(* CODESYS project ExtractAnyString.library
   Author: Piotr Pawlowski
   Version: 1.0.0.0
   Company: Marden Edwards
   Title: Extrac String
   Placeholder: EXTRACT
   LanguageModelAttribute: qualified-access-only
   DefaultNamespace: EXTRACT
   DocFormat: TcDocGen

Project tree, tasks and I/O mapping:
  libraries: Tc2_Standard, * (Beckhoff Automation GmbH); Tc2_System, * (Beckhoff Automation GmbH); Tc2_Utilities, * (Beckhoff Automation GmbH)
  DUTs/
    String/
      data type E_ExtrMode
      data type T_Char
      data type T_LongSTRING
  GVLs/
  POUs/
    String FB/
      function block FB_ExtractAnyString [ST]
      function block FB_ExtractString [ST]
    Strings FUN/
      function F_ReplaceLongSingleChar [ST]
  Version/
    global variables Global_Version
*)

// DUTs/String/E_ExtrMode
{attribute 'qualified_only'}
{attribute 'strict'}
TYPE E_ExtrMode :
(
	WITHIDENT,						//extract with ident and dont purge left side string
	WITHIDENT_PURGE,				//extract with ident and purge left side string
	WITHOUTIDENT,					//extract with ident and dont purge left side string, both ident left in origin string 
	WITHOUTIDENT_PURGE,				//extract with ident and purge left side string, only sufix ident left in origin string
	WITHOUTIDENT_REMIDENT,			//extract with ident and dont purge left side string, no ident left in origin string
	WITHOUTIDENT_REMIDENT_PURGE		//extract with ident and purge left side string, no ident left in origin string
);
END_TYPE

// DUTs/String/T_Char
TYPE T_Char : STRING[1];
END_TYPE

// DUTs/String/T_LongSTRING
TYPE T_LongSTRING : STRING(1023);
END_TYPE

// Version/Global_Version
{attribute 'TcGenerated'}
{attribute 'no-analysis'}
{attribute 'linkalways'}
// This function has been automatically generated from the project information.
VAR_GLOBAL CONSTANT
	{attribute 'const_non_replaced'}
	stLibVersion_Extrac_String : ST_LibVersion := (iMajor := 1, iMinor := 0, iBuild := 0, iRevision := 0, nFlags := 0, sVersion := '1.0.0.0');
END_VAR

// POUs/String FB/FB_ExtractAnyString
// Extracts a sub-string defined by prefix and suffix 
// Works in one cycle but as FB to not use stack memore due to LongString data defined
FUNCTION_BLOCK FB_ExtractAnyString
VAR_INPUT
	bExtractData			: BOOL;			(* set TRUE to remove prefix and suffix from strData *)
	nExtractChars			: UDINT;			(* if suffix is blank, number of data chars to extract *)
	sPrefix					: T_LongSTRING;	(* prefix string extended from T_MaxString to T_LongSTRING *)
	sSuffix					: T_LongSTRING;	(* suffix string extended from T_MaxString to T_LongSTRING *)
	bIgnoreCase				: BOOL;
	eExtractMode			: E_ExtrMode	:= E_ExtrMode.WITHOUTIDENT_REMIDENT;
	//bIncludeIdentifiers	: BOOL;
END_VAR
VAR_IN_OUT
	sDataString				: T_LongSTRING;	(* string to be searched *)
END_VAR
VAR_OUTPUT
	bStringFound			: BOOL;			(* TRUE = sub-string with matching prefix/suffix found *)
	sExtractedString		: T_LongSTRING;	(* extracted data *)
	nExtractedStringPos		: UDINT;			(* start pos of extracted string in strString *)
	nExtractedStringLen		: UDINT;
	nDataStringLen			: UDINT;
END_VAR
VAR
	
	//_rtExecute			: R_trig;
	
	_nExtractChars			: UDINT;
	_sPrefix				: T_LongSTRING;	(* prefix string *)
	_sSuffix				: T_LongSTRING;	(* suffix string *)
	_sDataString			: T_LongSTRING;	(* string to be searched *)
	
	_bIncludeIdentifiers	: BOOL;
	_bPurgeFullString		: BOOL;
	
	_nDataStringLen			: UDINT;
	_nPrefixLen				: UDINT;
	_nSuffixLen				: UDINT;
	
	_bPrefixFound			: BOOL;
	_bSuffixFound			: BOOL;
	
	_bPrefixIndex			: UDINT;
	_bTempSuffixIndex		: UDINT;
	_bSuffixIndex			: UDINT;
	
	_nStartDataPos			: UDINT;
	_nAbsolutDataPos		: UDINT;
	_nEndDataPos			: UDINT;
	_nExtractedDataLen		: UDINT;
	
	_nTerminatePos			: UDINT;
END_VAR

//	EXTRWITHIDENT						//extract with ident and dont purge left side string
//	EXTRWITHIDENT_PURGE					//extract with ident and purge left side string
//	EXTRWITHOUTIDENT					//extract with ident and dont purge left side string, both ident left in origin string 
//	EXTRWITHOUTIDENT_PURGE				//extract with ident and purge left side string, only sufix ident left in origin string
//	EXTRWITHOUTIDENT_REMIDENT			//extract with ident and dont purge left side string, no ident left in origin string
//	EXTRWITHOUTIDENT_REMIDENT_PURGE		//extract with ident and purge left side string, no ident left in origin string

//====================================================================================	
IF 	eExtractMode = E_ExtrMode.WITHIDENT 			OR 
	eExtractMode = E_ExtrMode.WITHIDENT_PURGE 	THEN
	
	_bIncludeIdentifiers	:= TRUE;
ELSE 
	_bIncludeIdentifiers	:= FALSE;
END_IF

IF 	eExtractMode = E_ExtrMode.WITHIDENT_PURGE 		OR 
	eExtractMode = E_ExtrMode.WITHOUTIDENT_PURGE 	OR 
	eExtractMode = E_ExtrMode.WITHOUTIDENT_REMIDENT_PURGE THEN
	
	_bPurgeFullString	:= LEN2(ADR(sDataString)) = SIZEOF(sDataString)-1;
ELSE 
	_bPurgeFullString	:= FALSE;
END_IF

//====================================================================================	

(* rising edge of bExecute *)
//_rtExecute(CLK := bExtractData);

//IF _rtExecute.Q THEN
	
//====================================================================================	
	bStringFound 		:= FALSE;
	
	_sDataString 		:= '';
	_sPrefix 			:= '';
	_sSuffix 			:= '';
	
	_bPrefixFound		:= FALSE;
	_bSuffixFound		:= FALSE;
		
	_bPrefixIndex		:= 0;
	_bSuffixIndex		:= 0;
		
	_nStartDataPos		:= 0;
	_nAbsolutDataPos	:= 0;
	_nEndDataPos		:= 0;
	//_ExtractedDataLen	:= 0;
	
	 (*calc string lengths *)
	_nDataStringLen 	:= LEN2(ADR(sDataString));
	_nPrefixLen 		:= LEN2(ADR(sPrefix));
	_nSuffixLen 		:= LEN2(ADR(sSuffix));
	
	_nExtractChars:= LIMIT(0, nExtractChars, _nDataStringLen);
	
	(*clear outputs*)
	nExtractedStringPos	:= 0;
	nExtractedStringLen	:= 0;
	nDataStringLen		:= _nDataStringLen;

//====================================================================================	
	
	(* matching for Prefix and Suffix is case-sesnsitive - worsk only with T_MaxString *)
	IF bIgnoreCase AND 
		_nDataStringLen < 256 	AND 
		_nPrefixLen < 256 		AND 
		_nSuffixLen < 256 		THEN
		
		(* internal comparators are all converted to lower case *)
		_sDataString 	:= F_ToLCase(sDataString);
		_sPrefix 		:= F_ToLCase(sPrefix);
		_sSuffix 		:= F_ToLCase(sSuffix);
		
	ELSE
		(* internal comparators are not changed *)
		_sDataString 	:= sDataString;
		_sPrefix 		:= sPrefix;
		_sSuffix 		:= sSuffix;
	END_IF

//====================================================================================	

	IF _nPrefixLen = 0 AND  _nExtractChars > 0 THEN
		
		_bPrefixIndex		:= 1;
		_nStartDataPos		:= 1;
		nExtractedStringPos := 1;
		
	ELSIF _nPrefixLen > 0 THEN		//if _nPrefixLen = 0 then _bPrefixIndex and _StartDataPos remains 0 from init state
		
		_bPrefixIndex	:= FIND2(ADR(_sDataString), ADR(_sPrefix));		//find search only if prefix declared on the input
	
		IF _bPrefixIndex > 0 THEN		//_bPrefixIndex as result form find can be onlu positive range
			
			_bPrefixFound := TRUE;		// _bPrefixFound guarantee _StartDataPos > 0
			_nStartDataPos 	:= SEL(_bIncludeIdentifiers, _bPrefixIndex + _nPrefixLen, _bPrefixIndex);
			_nAbsolutDataPos	:= _bPrefixIndex + _nPrefixLen;
			
			nExtractedStringPos := _nStartDataPos;
		END_IF
	END_IF	
	
//====================================================================================		

	IF _nSuffixLen = 0 AND  _nExtractChars > 0 THEN //IF only nExtractChars is declared THEN _EndDataPos pointing on elemnt determinated by nExtractChars or on last elemnt OF DataString
		
		_bSuffixIndex := _bPrefixIndex + _nPrefixLen + _nExtractChars;
		_nEndDataPos := MIN(_bSuffixIndex, _nDataStringLen);
		
		IF _nEndDataPos > _nStartDataPos THEN  // check if both pointers not point on last DataString elemnt
			_bSuffixFound := TRUE;	// _bSuffixFound guarantee _EndDataPos > 0 and found after _StartDataPos
		END_IF
		
	ELSIF _nSuffixLen > 0 THEN // if _nSuffixLen declared, then ignor nExtractChars and search for find sufix position using 
		
		// Include Sufix change shift if onle Prfix was found >> SEL(_bPrefixFound, 0, _StartDataPos - 1)
		_bTempSuffixIndex	:= FIND2(ADR(_sDataString) + SEL(_bPrefixFound, 0, _nAbsolutDataPos - 1), ADR(_sSuffix)); //find search only if sufix declared on the input and on index after prefix
		IF _bTempSuffixIndex > 0 THEN
			_bSuffixIndex	:= _bTempSuffixIndex + SEL(_bPrefixFound, 0, _nAbsolutDataPos - 1);	//Recalculate Sufix real position if sufix found or _bSuffixIndex remain 0 form init
		END_IF
		
		(*_bTempSuffixIndex gurantee that sufix was search after prefix position so _EndDataPos always greater than _StartDataPos *) 
		IF _bSuffixIndex > 0 THEN
			_bSuffixFound := TRUE;	// _bSuffixFound guarantee _EndDataPos > 0
			_nEndDataPos := SEL(_bIncludeIdentifiers,_bSuffixIndex, _bSuffixIndex + _nSuffixLen);
		END_IF
	END_IF
	
//====================================================================================		
	
	MEMSET(ADR(sExtractedString), 16#00, SIZEOF(sExtractedString));	//Clean sExtractedString area for new data

	IF _bPrefixFound AND _bSuffixFound THEN

		DELETE2(ADR(sDataString), ADR(sExtractedString), SIZEOF(sExtractedString), 
											SIZEOF(sExtractedString) - _nEndDataPos , _nEndDataPos);
		DELETE2(ADR(sExtractedString), ADR(sExtractedString), SIZEOF(sExtractedString), _nStartDataPos -1, 1);
		
	ELSIF _nPrefixLen = 0 AND _nSuffixLen = 0 AND _nExtractChars >= _nEndDataPos THEN		
		
		sExtractedString := sDataString;
		
	ELSIF _nPrefixLen = 0 AND _bSuffixFound THEN		// TO BE CONSIDERED IF WE WANT THIS CONDITION - IT WORKS LIKE LEFT
		
		_nStartDataPos := 1;
		DELETE2(ADR(sDataString), ADR(sExtractedString), SIZEOF(sExtractedString), 
										SIZEOF(sExtractedString) - _nEndDataPos , _nEndDataPos);
										
	ELSIF _bPrefixFound AND _nSuffixLen = 0 AND _nExtractChars = 0 THEN
		
		_nEndDataPos		:= _nDataStringLen;
		DELETE2(ADR(sDataString), ADR(sExtractedString), SIZEOF(sExtractedString), _nStartDataPos -1, 1);
		
	END_IF
		
	nExtractedStringLen	:= LEN2(ADR(sExtractedString));
	IF nExtractedStringLen <> 0 THEN  bStringFound := TRUE; END_IF
	
//====================================================================================
	IF NOT bStringFound AND _bPurgeFullString THEN
		
		sDataString := '';
		nDataStringLen := 0;
		
	ELSIF sExtractedString = sDataString THEN
		
		sDataString := '';
		nDataStringLen := 0;
		
	ELSIF bStringFound THEN //Terminate DataString only if endpositin for sufix is determinated and guratnee _EndDataPos greater then 0
		
		CASE eExtractMode OF

			E_ExtrMode.WITHIDENT:
			
				DELETE2(ADR(sDataString), ADR(sDataString), SIZEOF(sDataString), nExtractedStringLen, _nStartDataPos);		
					
			E_ExtrMode.WITHIDENT_PURGE:	
			
				IF _nEndDataPos = _nDataStringLen THEN
					DELETE2(ADR(sDataString), ADR(sDataString), SIZEOF(sDataString), _nEndDataPos, 1);
				ELSE
					DELETE2(ADR(sDataString), ADR(sDataString), SIZEOF(sDataString), _nEndDataPos -1, 1);
				END_IF
					
			E_ExtrMode.WITHOUTIDENT:		
			
				 DELETE2(ADR(sDataString), ADR(sDataString), SIZEOF(sDataString), nExtractedStringLen, _nStartDataPos);	
		
			E_ExtrMode.WITHOUTIDENT_PURGE:
						
				IF _nEndDataPos = _nDataStringLen THEN
					DELETE2(ADR(sDataString), ADR(sDataString), SIZEOF(sDataString), _nEndDataPos, 1);
				ELSE
					DELETE2(ADR(sDataString), ADR(sDataString), SIZEOF(sDataString), _nEndDataPos -1, 1);
				END_IF
				
			E_ExtrMode.WITHOUTIDENT_REMIDENT:
			
				DELETE2(ADR(sDataString), ADR(sDataString), SIZEOF(sDataString), 
										nExtractedStringLen + _nPrefixLen + _nSuffixLen, _bPrefixIndex);	
		
			E_ExtrMode.WITHOUTIDENT_REMIDENT_PURGE:		
						
				IF _nEndDataPos = _nDataStringLen THEN
					DELETE2(ADR(sDataString), ADR(sDataString), SIZEOF(sDataString), _nEndDataPos, 1);
				ELSE
					DELETE2(ADR(sDataString), ADR(sDataString), SIZEOF(sDataString), _bSuffixIndex + _nSuffixLen -1, 1);
				END_IF
				
		ELSE
			
			DELETE2(ADR(sDataString), ADR(sDataString), SIZEOF(sDataString), 
							nExtractedStringLen + _nPrefixLen + _nSuffixLen, _bPrefixIndex);
							
		END_CASE
	
		nDataStringLen := LEN2(ADR(sDataString));
	END_IF
//END_IF


(*

		
		IF _bSuffixIndex > _nDataStringLen THEN	//_EndDataPos cannot bi greater then _nDataStringLen due to previuse min condition
			_ExtractedDataLen := _EndDataPos -_StartDataPos + 1; // if _EndDataPos pointing on last element of sDataString, we must include it ofr extratcion
		ELSE
			_ExtractedDataLen := _EndDataPos -_StartDataPos;	//if prefix and sufix are found  _ExtractedDataLen always greater than 0
		END_IF
		
		MEMMOVE(ADR(sExtractedString),ADR(sDataString) + _StartDataPos -1 , _ExtractedDataLen);	// _StartDataPos -1 as initial adress has alredy value 1
		//MEMSET(ADR(sExtractedString) + _ExtractedDataLen, 16#00, _nDataStringLen - _ExtractedDataLen);
		
		
		
		//MEMMOVE(ADR(sExtractedString),ADR(sDataString), _EndDataPos);
		//MEMSET(ADR(sExtractedString) + _EndDataPos, 16#00, _nDataStringLen - _EndDataPos);
		
		
		
	
		IF _bSuffixIndex > _nDataStringLen THEN	//_EndDataPos cannot bi greater then _nDataStringLen due to previuse min condition
			_nTerminatePos := _EndDataPos;
		ELSE
			_nTerminatePos := SEL(_bIncludeIdentifiers, _EndDataPos + _nSuffixLen, _EndDataPos) -1; //sub 1 from final result as adressing of char start form pos 1
			//so if Terminate index should be 10 then _nTerminatePos must be 9 to add with initial addres of DataString
		END_IF
		
		IF _nDataStringLen > _nTerminatePos THEN	// guarantee we are not operating beyond DataString area
			MEMMOVE(ADR(sDataString), ADR(sDataString) + _nTerminatePos, _nDataStringLen - _nTerminatePos);
			MEMSET(ADR(sDataString) + _nDataStringLen - _nTerminatePos, 16#00, _nTerminatePos);
		ELSIF _nDataStringLen <= _nTerminatePos THEN
			sDataString := '';
		END_IF
			
	*)

END_FUNCTION_BLOCK

// POUs/String FB/FB_ExtractString
(* extracts a sub-string defined by prefix and suffix *)
FUNCTION_BLOCK FB_ExtractString
VAR_INPUT
	bExtractData		: BOOL;			(* set TRUE to remove prefix and suffix from strData *)
	nExtractChars		: UINT;			(* if suffix is blank, number of data chars to extract *)
	strPrefix			: T_MaxString;	(* prefix string *)
	strSuffix			: T_MaxString;	(* suffix string *)
END_VAR
VAR_IN_OUT
	strString			: T_MaxString;	(* string to be searched *)
END_VAR
VAR_OUTPUT
	bStringFound		: BOOL;			(* TRUE = sub-string with matching prefix/suffix found *)
	nStartPos			: UINT;			(* start pos of extracted string in strString *)
	strData				: T_MaxString;	(* extracted data *)
END_VAR
VAR
	nStringLen			: UINT;
	nPrefixLen			: UINT;
	nSuffixLen			: UINT;
	nEndPos				: UINT;
	bStartPosFound		: BOOL;
	bEndPosFound		: BOOL;
	nChars				: UINT;
	nMaxIndex			: UINT;
	nIndex				: UINT;
END_VAR
(*
-------------------------------------------------------------------------------------------------
DATE		Version	Author	Comments
-------------------------------------------------------------------------------------------------
30/01/2015	3.00.00	PB		bExtractData input added to specify whether prefix and suffix should be removed from strData
							bIgnoreCase input removed
							Major optimisation to reduce time taken to find a string

-------------------------------------------------------------------------------------------------
06/09/2012	1.41.00	PB		strData output added which returns strResult without the prefix and suffix
06/07/2011	1.23.00	PB		Pre-check added to ensure that strString is not empty
07/06/2011	1.19.00	PB		bIgnoreCase input added, set to TRUE to ignore upper/lower case when matching Prefix and Suffix
31/01/2011	1.08.03	PB		Bug fix - strings now handled correctly if strSuffix is longer than 1 char
							Search for suffix changed to start after prefix position
22/11/2010	1.07.01	PB		Initial release

-------------------------------------------------------------------------------------------------
*)

(* calc string lengths *)
nStringLen := INT_TO_UINT(LEN(strString));
nPrefixLen := INT_TO_UINT(LEN(strPrefix));
nSuffixLen := INT_TO_UINT(LEN(strSuffix));

(* string to be searched is not empty and prefix or suffix or no or chars to extract is defined *)
IF nStringLen > 0 AND (nPrefixLen > 0 OR nSuffixLen > 0 OR nExtractChars > 0) THEN

	(* clear outputs *)
	bStringFound := FALSE;
	nChars := 0;
	nStartPos := 0;
	strData := '';

	(* initialise char index values *)
	bStartPosFound := FALSE;
	bEndPosFound := FALSE;
	nEndPos := 0;

	(* max search index, based on string length - 1 due to starting at 0 and length of prefix *)
	nMaxIndex := (nStringLen - 1) + (nPrefixLen - 1);

	(* for each character in the string *)
	FOR nIndex := 0 TO nMaxIndex DO

		(* prefix has not been found *)
		IF bStartPosFound = FALSE THEN

			(* no prefix defined  *)
			IF nPrefixLen = 0 THEN

				(* start at beginning if string *)
				nStartPos := 1;
				bStartPosFound := TRUE;

			(* prefix defined  *)
			ELSE

				(* compare partial string with prefix *)
				IF MEMCMP(ADR(strString) + nIndex, ADR(strPrefix), nPrefixLen) = 0 THEN

					(* prefix position found *)
					nStartPos := nIndex + 1;
					bStartPosFound := TRUE;

					(* skip to end of prefix to continue search *)
					nIndex := nIndex + nPrefixLen - 1;
				END_IF
			END_IF

		(* suffix has not been found *)
		ELSIF bEndPosFound = FALSE THEN

			(* no suffix defined  *)
			IF nSuffixLen = 0 THEN

				(* start at 1st char of string *)
				bEndPosFound := TRUE;

				(* calculate end position *)
				nEndPos := MIN((nStartPos - 1) + nExtractChars + nPrefixLen, nStringLen);

			(* suffix defined  *)
			ELSE

				(* compare partial string with suffix *)
				IF MEMCMP(ADR(strString) + nIndex, ADR(strSuffix), nSuffixLen) = 0 THEN

					(* suffix position found, calculate end position *)
					nEndPos := nIndex + nSuffixLen;
					bEndPosFound := TRUE;

					(* no prefix defined and number of chars to extract is defined *)
					IF nPrefixLen = 0 AND nExtractChars > 0 THEN

						(* re-calculate start position *)
						nStartPos := MAX(nEndPos - nExtractChars - 1, 1);
					END_IF

					(* search complete, quit FOR loop *)
					EXIT;
				END_IF
			END_IF

		(* prefix and suffix found *)
		ELSE

			(* quit FOR loop *)
			EXIT;
		END_IF
	END_FOR

	(* start and end positions known *)
	IF bStartPosFound = TRUE AND bEndPosFound = TRUE THEN

		(* string has been found *)
		bStringFound := TRUE;

		(* return string without prefix and suffix *)
		IF bExtractData = TRUE THEN

			(* total chars to be moved to strData *)
			nChars := (nEndPos - (nStartPos - 1)) - nPrefixLen - nSuffixLen;

			(* 1 or more chars to be moved *)
			IF nChars > 0 THEN

				(* move data to strData *)
				MEMMOVE(ADR(strData), ADR(strString) + (nStartPos - 1) + nPrefixLen, nChars);
			END_IF

		(* return string with prefix and suffix *)
		ELSE

			(* total chars to be moved to strData *)
			nChars := nEndPos - (nStartPos - 1);

			(* 1 or more chars to be moved *)
			IF nChars > 0 THEN

				(* move data to strData *)
				MEMMOVE(ADR(strData), ADR(strString) + (nStartPos - 1), nChars);
			END_IF
		END_IF

		(* terminate strData *)
		MEMSET(ADR(strData) + nChars, 16#00, 1);

		(* 1 or more chars after strSuffix *)
		IF nStringLen > (nEndPos - (nStartPos - 1)) THEN

			(* shift post-suffix chars to prefix position *)
			MEMMOVE(ADR(strString) + (nStartPos - 1), ADR(strString) + nEndPos, nStringLen - (nEndPos - (nStartPos - 1)));
		END_IF

		(* terminate strString *)
		MEMSET(ADR(strString) + nStringLen - (nEndPos - (nStartPos - 1)), 16#00, 1);
	END_IF

(* string to be searched is empty or prefix and suffix and both blank *)
ELSE

	(* clear outputs *)
	bStringFound := FALSE;
	nChars := 0;
	strData := '';
END_IF

END_FUNCTION_BLOCK

// POUs/Strings FUN/F_ReplaceLongSingleChar
FUNCTION F_ReplaceLongSingleChar : T_LongSTRING
VAR_INPUT
	sFullCode		: T_LongSTRING;
	sCharRemove			: T_Char := '$1D';
	sReplacmentChar		: T_Char := '';
END_VAR
VAR
	sCodeSize		: STRING;
END_VAR

WHILE FIND2(ADR(sFullCode), ADR(sCharRemove)) > 0 DO
	REPLACE2(ADR(sFullCode),ADR(sReplacmentChar), ADR(sFullCode), 
						SIZEOF(sFullCode), LEN2(ADR(sCharRemove)), FIND2(ADR(sFullCode), ADR(sCharRemove)));
END_WHILE

(*Diagnostic part for long stirng operation *)
//sCodeSize := TO_STRING(LEN2(ADR(sFullCode)));
//CONCAT2(ADR(sCodeSize), ADR('_'), ADR(sCodeSize), SIZEOF(sCodeSize));	
//INSERT2(ADR(sFullCode), ADR(sCodeSize), ADR(sFullCode), SIZEOF(sFullCode), 0);
	
F_ReplaceLongSingleChar	:= sFullCode;

END_FUNCTION
